(* IEC 61131-3 sources: CodesysTest/alpha/export/FBs/Components/BagOpenFingersFB.pou, 3 files *)

(* ---- BagOpenFingersFB.pou.st ---- *)
(*#-#-#-#-#-#-#-#-#-#---Declaration---#-#-#-#-#-#-#-#-#-#-#-#-#*)

FUNCTION_BLOCK BagOpenFingersFB EXTENDS BaseComponentFB
VAR_INPUT

END_VAR
VAR_IN_OUT

END_VAR
VAR_OUTPUT
    releaseOutput : BOOL;
	grabOutput : BOOL;
END_VAR
VAR
    _releaseCommand : BOOL;
    _grabCommand : BOOL;
END_VAR
(*#-#-#-#-#-#-#-#-#-#---Implementation---#-#-#-#-#-#-#-#-#-#-#-#-#*)

SUPER^();
releaseOutput := _releaseCommand AND enable;
grabOutput := _grabCommand AND enable;

(* ---- Grab.m.st ---- *)
(*#-#-#-#-#-#-#-#-#-#---Declaration---#-#-#-#-#-#-#-#-#-#-#-#-#*)

METHOD Grab
VAR_INPUT
END_VAR
(*#-#-#-#-#-#-#-#-#-#---Implementation---#-#-#-#-#-#-#-#-#-#-#-#-#*)

_releaseCommand := FALSE;
_grabCommand := TRUE;
HMIData.bagOpenFingerCycles.Increment();

(* ---- Release.m.st ---- *)
(*#-#-#-#-#-#-#-#-#-#---Declaration---#-#-#-#-#-#-#-#-#-#-#-#-#*)

METHOD Release
VAR_INPUT
END_VAR
(*#-#-#-#-#-#-#-#-#-#---Implementation---#-#-#-#-#-#-#-#-#-#-#-#-#*)

_releaseCommand := TRUE;
_grabCommand := FALSE;
